FUNCTION_BLOCK FB_WriteFile

VAR_INPUT 
	InDirFile : STRING(1000);
	InAmsId : T_AmsNetID :='';
	InPMessage: POINTER TO BYTE;
	InLMessage: UDINT;
	InStart : BOOL;
	InMode : DWORD := 16#4;	// Append Mode . 
END_VAR

VAR_OUTPUT
	OutBusy 	: BOOL;
	OutError 	: BOOL;
	OutErrorId 	: STRING;
	cbWritten 	: UDINT;
	OutCompleted : BOOL;
END_VAR

VAR 
MesDataExd: LoggerCSV;
	FileHandle 	: UINT;
	select		: INT;
	AX_ErrorId	: ARRAY[1..NbSteps] OF UDINT;
	AX_Error 	: ARRAY[1..NbSteps] OF BOOL;
	OpenFile 	: FB_FileOpen;
	CloseFile 	: FB_FileClose;
	WriteFile 	: FB_FileWrite;
	TextToWrite : STRING(255);
	nSeekPos 	: DINT;
	i 			: UINT;
	bCompleted	: BOOL;
	Trigger		: R_TRIG;
END_VAR

VAR CONSTANT
	NbSteps 	: UINT := 3;
END_VAR

OutCompleted := FALSE;
CASE select OF
	0: // Initialize
		Trigger(CLK := InStart);
		IF Trigger.Q THEN
			select := 1;
			OutBusy := TRUE;
			OutError := FALSE;
			OutErrorId :='';
		END_IF
	1:
		OpenFile(sNetId := InAmsId, 
			sPathName := InDirFile,
			nMode := InMode,
			ePath := Path_generic,
			bExecute := TRUE,
			hFile => FileHandle,
			nErrId => AX_ErrorId[Select],
			bError => AX_Error[Select]
		);
		IF NOT(OpenFile.bBusy) THEN
 			IF NOT(OpenFile.bError) THEN
				select := select+1;
				OpenFile(bExecute := FALSE);
			ELSE
				select := -1;
			END_IF
		END_IF

	2: 
		WriteFile(
			sNetId := InAmsId,
			hFile := FileHandle,
			pWriteBuff := InPMessage,
			cbWriteLen := InLMessage,
			bExecute := TRUE,
			nErrId => AX_ErrorId[Select],
			bError => AX_Error[Select]
		);
		IF NOT(WriteFile.bBusy) THEN
			IF NOT(WriteFile.bError) THEN
				select := select+1;
				WriteFile(bExecute := FALSE);
				cbWritten := WriteFile.cbWrite;
			ELSE
				select := -1;
			END_IF
		END_IF
	3 : 
		CloseFile(sNetId := InAmsId, 
			hFile := FileHandle,
			bExecute := TRUE, 
			tTimeout := T#1S,
			nErrId => AX_ErrorId[Select],
			bError => AX_Error[Select]
		);
		IF NOT(CloseFile.bBusy) THEN
			IF NOT(CloseFile.bError) THEN
				select := 10;
				CloseFile(bExecute := FALSE);
			ELSE
				select := -1;
			END_IF
		END_IF
		
	10: 
		FileHandle := 0;
		OutBusy := FALSE;
		select := 0;
		OutCompleted := TRUE;
		FOR i := 1 TO NbSteps DO
			AX_ErrorId[i] := 0;
			AX_Error[i] := FALSE;
		END_FOR
		
	-1 : 
		IF FileHandle <> 0 THEN
			CloseFile(sNetId := InAmsId, hFile := FileHandle, bExecute := TRUE);
		END_IF
		OpenFile(bExecute := FALSE);
		WriteFile(bExecute := FALSE);
		IF NOT(CloseFIle.bBusy) THEN
			CloseFile(bExecute := FALSE);
		END_IF
		M_AlarmManager();
		select := 10;
END_CASE

METHOD M_AlarmManager : BOOL
VAR
	j : UINT;
	StringInterm : STRING;
END_VAR
OutError := FALSE;
OutErrorId :='';
FOR j := 1 TO NbSteps DO
	OutError := OutError OR AX_Error[j];
	IF AX_Error[j] THEN
		OutErrorId := concat(concat(Concat(UINT_TO_STRING(j),'_'), UDINT_TO_STRING(AX_ERRORID[j])), CONCAT('*',OutErrorId));
	END_IF
END_FOR
END_METHOD

END_FUNCTION_BLOCK

(* stored: Version 1.1.0.1, ProductVersion 3.1.4024.6
   POU FB_WriteFile: Id {de6635fe-4006-4163-b280-71c930aab15b}, SpecialFunc None
   Method M_AlarmManager: Id {b7d49c4c-ab79-4989-8df5-eecf68676b70} *)
